TYPE ST_Child EXTENDS ST_Base : STRUCT
    fValue : REAL;
END_STRUCT
END_TYPE

(* stored: Version 1.1.0.1
   DUT ST_Child: Id {55555555-5555-5555-5555-555555555503} *)
